{attribute 'GeneratedUsingTerminal: EL6201-0000-0017'}
{attribute addProperty BoxType "EL6201-0000-0017"}
{attribute addProperty Id "Slave_15A_DO0BOOL1Slave_15A_DO1BOOL1Slave_15A_DO2BOOL1Slave_15A_DO3BOOL1Slave_15B_DO0BOOL1Slave_15B_DO1BOOL1Slave_15B_DO2BOOL1Slave_15B_DO3BOOL1"}
{attribute addProperty CRC "2675248977"}
{attribute addProperty Size "8"}
TYPE Slave_15_Outputs_9F750F51 :
STRUCT
	{attribute addProperty Name "Slave_15A_DO0"}
	Slave_15A_DO0 : BOOL;
	{attribute addProperty Name "Slave_15A_DO1"}
	Slave_15A_DO1 : BOOL;
	{attribute addProperty Name "Slave_15A_DO2"}
	Slave_15A_DO2 : BOOL;
	{attribute addProperty Name "Slave_15A_DO3"}
	Slave_15A_DO3 : BOOL;
	{attribute addProperty Name "Slave_15B_DO0"}
	Slave_15B_DO0 : BOOL;
	{attribute addProperty Name "Slave_15B_DO1"}
	Slave_15B_DO1 : BOOL;
	{attribute addProperty Name "Slave_15B_DO2"}
	Slave_15B_DO2 : BOOL;
	{attribute addProperty Name "Slave_15B_DO3"}
	Slave_15B_DO3 : BOOL;
END_STRUCT
END_TYPE

(* stored: Version 1.2.0.0, ProductVersion 3.1.4024.9
   DUT Slave_15_Outputs_9F750F51: Id {3efcf745-70c6-4eef-a5b6-6c015afcfb57} *)
